Omron Sysmac Studio project 교육자료_30_상수 제거_1 (Sysmac Studio 1.23.0.14, StandardProject)

# Controller new_Controller_0: NJ301-1100 version 1.9
Units and slaves: 전원 : NJ-Px3001; CPU : NJ301-1100; 0 : CJ1W-ID231 (J01); 1 : CJ1W-OD231 (J02)
Task PrimaryTask (priority 4, period or condition 1000): Program0

TYPE ENUM_O : (i_CY1 := 0, i_CY2N := 1, i_CY2P := 2, i_CY3 := 3, i_CY5 := 4, i_MT1P := 5); END_TYPE

VAR_GLOBAL
    cy10 : BOOL;  (* 공급실린더후진; at IOBus://rack#0/slot#0/Ch1_In/Ch1_In00 *)
    cy11 : BOOL;  (* 공급실린더전진; at IOBus://rack#0/slot#0/Ch1_In/Ch1_In01 *)
    cy12 : BOOL;  (* 재료공급확인_광센서; at IOBus://rack#0/slot#0/Ch1_In/Ch1_In02 *)
    cy20 : BOOL;  (* 송출실린더후진; at IOBus://rack#0/slot#0/Ch1_In/Ch1_In03 *)
    cy21 : BOOL;  (* 송출실린더전진; at IOBus://rack#0/slot#0/Ch1_In/Ch1_In04 *)
    cy30 : BOOL;  (* 송출실린더상승; at IOBus://rack#0/slot#0/Ch1_In/Ch1_In05 *)
    cy31 : BOOL;  (* 송출실린더하강; at IOBus://rack#0/slot#0/Ch1_In/Ch1_In06 *)
    cy40 : BOOL;  (* 정지실린더상승; at IOBus://rack#0/slot#0/Ch1_In/Ch1_In07 *)
    cy41 : BOOL;  (* 정지실린더하강; at IOBus://rack#0/slot#0/Ch1_In/Ch1_In08 *)
    cy42 : BOOL;  (* 정지위치확인_광센서; at IOBus://rack#0/slot#0/Ch1_In/Ch1_In09 *)
    cy51 : BOOL;  (* 흡착센서; at IOBus://rack#0/slot#0/Ch1_In/Ch1_In10 *)
    mt11 : BOOL;  (* 유도형센서; at IOBus://rack#0/slot#0/Ch1_In/Ch1_In11 *)
    mt12 : BOOL;  (* 용량형센서; at IOBus://rack#0/slot#0/Ch1_In/Ch1_In12 *)
    mt2Lccw : BOOL;  (* 적재함_리미트CCW; at IOBus://rack#0/slot#0/Ch1_In/Ch1_In13 *)
    mt2Pos1 : BOOL;  (* 적재함_Pos1; at IOBus://rack#0/slot#0/Ch1_In/Ch1_In14 *)
    mt2Pos2 : BOOL;  (* 적재함_Pos2; at IOBus://rack#0/slot#0/Ch1_In/Ch1_In15 *)
    mt2Lcw : BOOL;  (* 적재함_리미트CW; at IOBus://rack#0/slot#0/Ch2_In/Ch2_In01 *)
    mt2En : BOOL;  (* 적재함_엔코더; at IOBus://rack#0/slot#0/Ch2_In/Ch2_In02 *)
    pb1 : BOOL;  (* 푸쉬버튼1; at IOBus://rack#0/slot#0/Ch2_In/Ch2_In03 *)
    pb2 : BOOL;  (* 푸쉬버튼2; at IOBus://rack#0/slot#0/Ch2_In/Ch2_In04 *)
    pb3 : BOOL;  (* 푸쉬버튼3; at IOBus://rack#0/slot#0/Ch2_In/Ch2_In05 *)
    CY1 : BOOL;  (* 공급전후진Sol; at IOBus://rack#0/slot#1/Ch1_Out/Ch1_Out00 *)
    CY2N : BOOL;  (* 송출후진Sol; at IOBus://rack#0/slot#1/Ch1_Out/Ch1_Out01 *)
    CY2P : BOOL;  (* 송출전진Sol; at IOBus://rack#0/slot#1/Ch1_Out/Ch1_Out02 *)
    CY3 : BOOL;  (* 송출상승_하강Sol; at IOBus://rack#0/slot#1/Ch1_Out/Ch1_Out03 *)
    CY4 : BOOL;  (* 정지상승_하강Sol; at IOBus://rack#0/slot#1/Ch1_Out/Ch1_Out04 *)
    CY5 : BOOL;  (* 흡착전후진Sol; at IOBus://rack#0/slot#1/Ch1_Out/Ch1_Out05 *)
    MT1N : BOOL;  (* 컨베이어CCW; at IOBus://rack#0/slot#1/Ch1_Out/Ch1_Out06 *)
    MT1P : BOOL;  (* 컨베이어CW; at IOBus://rack#0/slot#1/Ch1_Out/Ch1_Out07 *)
    MT2N : BOOL;  (* 적재함CCW; at IOBus://rack#0/slot#1/Ch1_Out/Ch1_Out08 *)
    MT2P : BOOL;  (* 적재함CW; at IOBus://rack#0/slot#1/Ch1_Out/Ch1_Out09 *)
    LP1 : BOOL;  (* 적색램프; at IOBus://rack#0/slot#1/Ch1_Out/Ch1_Out10 *)
    LP2 : BOOL;  (* 녹색램프; at IOBus://rack#0/slot#1/Ch1_Out/Ch1_Out11 *)
    LP3 : BOOL;  (* 황색램프; at IOBus://rack#0/slot#1/Ch1_Out/Ch1_Out12 *)
    mt2Pos3 : BOOL;  (* 적재함_Pos3; at IOBus://rack#0/slot#0/Ch2_In/Ch2_In00 *)
END_VAR

PROGRAM Program0
VAR
    iaSeq : ARRAY[0..10] OF int;  (* 이동상태번호 매개변수 *)
    t1 : TON;  (* 0.35초 지연 *)
    c1 : CTU;  (* 3회 카운트 *)
    m102 : BOOL;  (* PB1 자기유지 메모리 *)
    temp : INT;  (* 임시 카운터값 표시 *)
    baRoot : ARRAY[0..10] OF bool;  (* 입력조건상태 매개변수 *)
    ba분류기_출력상태 : ARRAY[0..10,0..5] OF bool;  (* 출력상태번호 매개변수 *)
    J01 : CNT_LUT;  (* 순차회로 FB *)
    baJ01Out : ARRAY[0..5] OF bool;  (* FB출력 *)
    iJ01Seq : INT;  (* FB내부 동작번호 *)
    idx : DINT;
END_VAR
VAR_EXTERNAL
    pb1 : BOOL;
    LP1 : BOOL;
    LP2 : BOOL;
    pb2 : BOOL;
    pb3 : BOOL;
    LP3 : BOOL;
    cy10 : BOOL;
    cy11 : BOOL;
    cy12 : BOOL;
    cy20 : BOOL;
    cy21 : BOOL;
    cy30 : BOOL;
    cy31 : BOOL;
    cy40 : BOOL;
    cy41 : BOOL;
    cy42 : BOOL;
    cy51 : BOOL;
    mt11 : BOOL;
    mt12 : BOOL;
    mt2Lccw : BOOL;
    mt2Pos1 : BOOL;
    mt2Pos2 : BOOL;
    mt2Pos3 : BOOL;
    mt2Lcw : BOOL;
    mt2En : BOOL;
    CY1 : BOOL;
    CY2N : BOOL;
    CY2P : BOOL;
    CY3 : BOOL;
    CY4 : BOOL;
    CY5 : BOOL;
    MT1N : BOOL;
    MT1P : BOOL;
    MT2N : BOOL;
    MT2P : BOOL;
END_VAR

(* Section Section0: ladder, written here as Structured Text *)

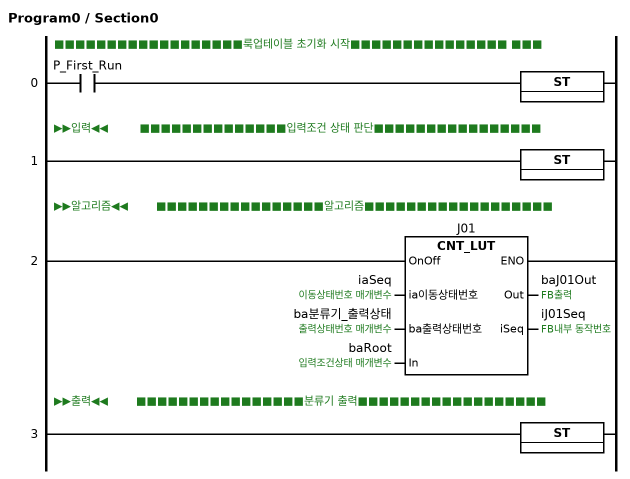
(* Rung 0: ■■■■■■■■■■■■■■■■■■룩업테이블 초기화 시작■■■■■■■■■■■■■■■ ■■■ *)
IF P_First_Run THEN
    
END_IF;
(* Rung 1: ▶▶입력◀◀         ■■■■■■■■■■■■■■입력조건 상태 판단■■■■■■■■■■■■■■■■ *)

(* Rung 2: ▶▶알고리즘◀◀        ■■■■■■■■■■■■■■■■알고리즘■■■■■■■■■■■■■■■■■■ *)
J01(OnOff := TRUE, ia이동상태번호 := iaSeq, ba출력상태번호 := ba분류기_출력상태, In := baRoot, Out => baJ01Out, iSeq => iJ01Seq);
(* Rung 3: ▶▶출력◀◀        ■■■■■■■■■■■■■■■■분류기 출력■■■■■■■■■■■■■■■■■■ *)

END_PROGRAM

FUNCTION_BLOCK CNT_LUT
VAR
    index : INT;
END_VAR
VAR_INPUT
    OnOff : BOOL;
    ia이동상태번호 : ARRAY[0..10] OF int;
    ba출력상태번호 : ARRAY[0..10,0..5] OF bool;
    In : ARRAY[0..10] OF bool;
END_VAR
VAR_OUTPUT
    Out : ARRAY[0..5] OF bool;
    iSeq : INT;
END_VAR
VAR_EXTERNAL
    cy10 : BOOL;
    cy12 : BOOL;
    cy11 : BOOL;
    cy42 : BOOL;
    cy31 : BOOL;
    cy30 : BOOL;
    cy51 : BOOL;
    cy21 : BOOL;
    cy20 : BOOL;
END_VAR
//	■■■■■■■■■■■■■■■■■■■■■■■■■■■■■■■■■■■■■■■■■■■■■■■■■■■■■■■■■
// ■■■■■■■■■■■■■■■■■■■■[ 분류기 펑션블록 (CNT_LUT 내용 ]■■■■■■■■■■■■■■■■■■■■■■		
//	■■■■■■■■■■■■■■■■■■■■■■■■■■■■■■■■■■■■■■■■■■■■■■■■■■■■■■■■■


//■알고리즘■ 분류기 회로 실행문 (분기문)
IF In[iSeq] THEN // abSeq ( 입력조건 상태) 에 따른 wSeq 값 이동 ( 일반 상태 및 금속의 경우 )
		iSeq := ia이동상태번호[iSeq]; 
END_IF;



// ■출력■ 분류기 회로 출력문
FOR index:=0 TO 5 BY 1 DO
	Out[index] := ba출력상태번호[iSeq, index];  
END_FOR;
END_FUNCTION_BLOCK